(* IEC 61131-3 sources: AcpTrakStarwheel/ (part 2) *)

(* ---- StarRecovery.st ---- *)
FUNCTION_BLOCK slStarRecovery

    CASE Internal.State OF

        slREC_STATE_IDLE:
            // ----------------------------------------------------------------------- disabled

            IF Enable THEN
                Busy := 1;
                Internal.OldRemainingCount := 0;
                IF Handle = 0 THEN
                    Error := 1;
                    ErrorID := slERR_INVALID_HANDLE;
                    Internal.State := slREC_STATE_ERROR;
                ELSE
                    Internal.Handle := Handle;
                    StarInternal ACCESS Internal.Handle;
                    IF StarInternal.TypeID <> slSTAR_INTERNAL_TYPE_ID THEN
                        Error := 1;
                        ErrorID := slERR_INVALID_HANDLE;
                        Internal.State := slREC_STATE_ERROR;
                    ELSE
                        brsmemset(ADR(Internal.Data), 0, SIZEOF(Internal.Data));
                        Internal.AsmGetInfo.Assembly    := ADR(Assembly);
                        Internal.AsmGetInfo.Execute     := TRUE;
                        Internal.State := slREC_STATE_CHECK_SECTOR_SIM;
                    END_IF
                END_IF
            END_IF

        slREC_STATE_CHECK_SECTOR_SIM:

            IF Internal.AsmGetInfo.Done THEN
                Internal.SecGetShuttle.Sector := ADR(Sector);
                Internal.SecGetShuttle.Mode := mcACPTRAK_SEARCH_BACKWARD;
                Internal.SecGetShuttle.Enable := TRUE;
                Internal.State := slREC_STATE_GET_SHUTTLES;
            ELSIF Internal.AsmGetInfo.Error THEN
                Internal.AsmGetInfo.Execute := FALSE;
                Error   := TRUE;
                ErrorID := Internal.AsmGetInfo.ErrorID;
                Internal.State := slREC_STATE_ERROR;
            END_IF;

        slREC_STATE_GET_SHUTTLES:
            // ----------------------------------------------------------------------- Get shuttles in sector

            IF NOT Enable THEN
                Internal.SecGetShuttle.Next := 0;
                Internal.SecGetShuttle.Enable := 0;
                Internal.State := slREC_STATE_WAIT_NOT_BUSY;
            ELSIF Internal.SecGetShuttle.Error THEN
                Internal.SecGetShuttle.Next := 0;
                Internal.SecGetShuttle.Enable := 0;
                Error := 1;
                ErrorID := Internal.SecGetShuttle.ErrorID;
                Internal.State := slREC_STATE_ERROR;
            ELSIF Internal.SecGetShuttle.Valid AND ((Internal.SecGetShuttle.RemainingCount <> Internal.OldRemainingCount) OR (Internal.SecGetShuttle.TotalCount <= 1)) THEN
                Internal.SecGetShuttle.Next := 0;
                IF Internal.SecGetShuttle.TotalCount > 0 THEN
                    Internal.Data.Init.ShuttlePos[Internal.Data.Init.NumShuttles] := Internal.SecGetShuttle.AdditionalInfo.Position;
                    Internal.Data.Init.ShuttleAxis[Internal.Data.Init.NumShuttles] := Internal.SecGetShuttle.Axis;
                    Internal.Data.Init.NumShuttles := Internal.Data.Init.NumShuttles + 1;
                    IF Internal.AsmGetInfo.AssemblyInfo.SimulationOnPlcMode = mcACPTRAK_SIM_STATE_OFF THEN
                        Internal.State := slREC_STATE_GET_SHUTTLES_NEXT;
                    ELSIF Internal.AsmGetInfo.AssemblyInfo.SimulationOnPlcMode = mcACPTRAK_SIM_STATE_ON THEN
                        Internal.RoutedMoveAbs.Sector   := ADR(Sector);
                        Internal.RoutedMoveAbs.Axis     := ADR(Internal.SecGetShuttle.Axis);
                        Internal.RoutedMoveAbs.Position := Internal.SecGetShuttle.AdditionalInfo.Position;
                        Internal.RoutedMoveAbs.Velocity := 1.0;
                        Internal.RoutedMoveAbs.Acceleration := 20.0;
                        Internal.RoutedMoveAbs.Deceleration := 20.0;
                        Internal.RoutedMoveAbs.AdvancedParameters.StartDirection    := mcDIR_UNDEFINED;
                        Internal.RoutedMoveAbs.AdvancedParameters.EndDirection      := mcDIR_UNDEFINED;
                        Internal.RoutedMoveAbs.AdvancedParameters.ShuttleOrientation    := mcDIR_UNDEFINED;
                        Internal.RoutedMoveAbs.Execute  := TRUE;

                        Internal.State  := slREC_STATE_ATTACH_TO_SECTOR;
                    END_IF;
                ELSE //No shuttles on the sector
                    Internal.SecGetShuttle.Enable := FALSE;
                    Internal.State := slREC_STATE_DONE;
                END_IF
            END_IF

        slREC_STATE_ATTACH_TO_SECTOR:

            IF Internal.RoutedMoveAbs.Done THEN
                Internal.RoutedMoveAbs.Execute  := FALSE;
                Internal.State  := slREC_STATE_GET_SHUTTLES_NEXT;
            ELSIF Internal.RoutedMoveAbs.Error THEN
                Internal.RoutedMoveAbs.Execute  := FALSE;
                Error   := TRUE;
                ErrorID := Internal.RoutedMoveAbs.ErrorID;
                Internal.State := slREC_STATE_ERROR;
            END_IF;

        slREC_STATE_GET_SHUTTLES_NEXT:
            // -----------------------------------------------------------------------

            IF NOT Enable THEN
                Internal.SecGetShuttle.Enable := 0;
                Internal.State := slREC_STATE_WAIT_NOT_BUSY;
            ELSIF Internal.SecGetShuttle.Error THEN
                Internal.SecGetShuttle.Enable := 0;
                Error := 1;
                ErrorID := Internal.SecGetShuttle.ErrorID;
                Internal.State := slREC_STATE_ERROR;
            ELSIF Internal.SecGetShuttle.Valid THEN
                IF Internal.SecGetShuttle.RemainingCount > 0 THEN
                    Internal.OldRemainingCount := Internal.SecGetShuttle.RemainingCount;
                    Internal.SecGetShuttle.Next := TRUE;
                    Internal.State := slREC_STATE_GET_SHUTTLES;
                ELSE
                    Internal.SecGetShuttle.Enable := FALSE;
                    Internal.State := slREC_STATE_GET_USERDATA;
                END_IF
            END_IF

        slREC_STATE_RELEASE_ZONE_CHECK:
            // ----------------------------------------------------------------------- Find shuttles in the release zone

            IF Enable THEN
                IF Internal.Data.Init.ShuttlePos[Internal.Data.Init.ShuttleEvalCount] >= Parameters.MeshZoneEndPos THEN
                    Internal.State := slREC_STATE_RELEASE_ZONE_RESIZE;
                ELSE //Go to next section
                    Internal.State := slREC_STATE_MESH_ZONE_CHECK;
                END_IF;
            ELSE
                Internal.State := slREC_STATE_WAIT_NOT_BUSY;
            END_IF

        slREC_STATE_RELEASE_ZONE_RESIZE:
            // -----------------------------------------------------------------------

            IF Enable THEN
                Internal.ShResize.Axis := ADR(Internal.Data.Init.ShuttleAxis[Internal.Data.Init.ShuttleEvalCount]);
                Internal.ShResize.Command := mcACPTRAK_RESIZE_DIMENSIONS;
                Internal.ShResize.ResizeParameter := Parameters.ResizeEnd;
                Internal.ShResize.Execute := TRUE;
                Internal.State := slREC_STATE_RELEASE_ZONE_SEND;
            ELSE
                Internal.State := slREC_STATE_WAIT_NOT_BUSY;
            END_IF

        slREC_STATE_RELEASE_ZONE_SEND:
            // -----------------------------------------------------------------------

            IF NOT Enable THEN
                Internal.ShResize.Execute := 0;
                Internal.State := slREC_STATE_WAIT_NOT_BUSY;
            ELSIF Internal.ShResize.Error THEN
                Internal.ShResize.Execute := 0;
                Error := 1;
                ErrorID := Internal.ShResize.ErrorID;
                Internal.State := slREC_STATE_ERROR;
            ELSIF Internal.ShResize.Done THEN
                Internal.RoutedMoveVel.Axis := ADR(Internal.Data.Init.ShuttleAxis[Internal.Data.Init.ShuttleEvalCount]);
                Internal.RoutedMoveVel.Sector := ADR(Parameters.Release.DestinationSector);
                Internal.RoutedMoveVel.Velocity := Parameters.Release.Velocity;
                Internal.RoutedMoveVel.Acceleration := Parameters.Release.Acceleration;
                Internal.RoutedMoveVel.Deceleration := Parameters.Release.Deceleration;
                Internal.RoutedMoveVel.AdvancedParameters.StartDirection    := mcDIR_POSITIVE;
                Internal.RoutedMoveVel.AdvancedParameters.EndDirection      := mcDIR_UNDEFINED;
                Internal.RoutedMoveVel.AdvancedParameters.ShuttleOrientation    := mcDIR_UNDEFINED;

                Internal.RoutedMoveVel.Execute := TRUE;
                Internal.Data.Init.ShuttleEvalCount := Internal.Data.Init.ShuttleEvalCount + 1;
                Internal.State := slREC_STATE_RELEASE_ZONE_NEXT;
            END_IF;

        slREC_STATE_RELEASE_ZONE_NEXT:
            // ----------------------------------------------------------------------- See if there are anymore shuttles to recover

            IF NOT Enable THEN
                Internal.RoutedMoveVel.Execute := 0;
                Internal.State := slREC_STATE_WAIT_NOT_BUSY;
            ELSIF Internal.RoutedMoveVel.Error THEN
                Internal.RoutedMoveVel.Execute := 0;
                Error := 1;
                ErrorID := Internal.RoutedMoveVel.ErrorID;
                Internal.State := slREC_STATE_ERROR;
            ELSIF Internal.RoutedMoveVel.Active THEN
                Internal.RoutedMoveVel.Execute := FALSE;
                IF Internal.Data.Init.ShuttleEvalCount < Internal.Data.Init.NumShuttles THEN
                    Internal.State := slREC_STATE_RELEASE_ZONE_CHECK;
                ELSE
                    Internal.State := slREC_STATE_DONE;
                END_IF;
            END_IF

        slREC_STATE_MESH_ZONE_CHECK:
            // ----------------------------------------------------------------------- Find shuttles in the sync zone

            IF Enable THEN
                IF Internal.Data.Init.ShuttlePos[Internal.Data.Init.ShuttleEvalCount] < Parameters.MeshZoneEndPos AND
                    Internal.Data.Init.ShuttlePos[Internal.Data.Init.ShuttleEvalCount] >= (Parameters.MeshZoneStartPos) THEN
                    Internal.State := slREC_STATE_MESH_ZONE_TARGET;
                ELSE
                    //IF Parameters.SyncFurtherInEnabled THEN
                    //    Internal.Data.Sync.PocketEvalIndex    := ClosestSyncPocket(Parameters.MeshZoneStartPos, Parameters.ProcessPointStartPosition + Parameters.StartOffset, Internal.Handle);
                   // END_IF;
                    Internal.State := slREC_STATE_SYN_ZONE_CHECK;
                END_IF
            ELSE
                Internal.State := slREC_STATE_WAIT_NOT_BUSY;
            END_IF

        slREC_STATE_MESH_ZONE_TARGET:
            // ----------------------------------------------------------------------- Find the closest pocket to it and see if it is in tolerance

            //TODO: Replace with function
            //Find the closest pocket to to the shuttle
            StarInternal ACCESS Internal.Handle;
            Internal.Data.Mesh.PocketEvalIndex  := 0;
            Internal.Data.Mesh.PocketEvalIndexValid := FALSE;
            Internal.Data.Mesh.NextClosestPocketIndex   := 0;
            IF StarInternal.MaxTargetIndex > 0 THEN
                FOR Internal.i := 0 TO StarInternal.MaxTargetIndex DO
                    Internal.Data.Mesh.ShuttleErrorNew := StarInternal.PocketSync[Internal.i].TargetPosition - Internal.Data.Init.ShuttlePos[Internal.Data.Init.ShuttleEvalCount];
                    IF Internal.i = 0 THEN
                        Internal.Data.Mesh.ShuttleError := Internal.Data.Mesh.ShuttleErrorNew;
                        Internal.Data.Mesh.NextClosestPocketError := StarInternal.PocketSync[1].TargetPosition - Internal.Data.Init.ShuttlePos[Internal.Data.Init.ShuttleEvalCount];
                        Internal.Data.Mesh.NextClosestPocketIndex   := 1;
                    END_IF;
                    //Ignore any pockets that are before the sync zone
                    IF StarInternal.PocketSync[Internal.i].TargetPosition >= Parameters.ProcessPointStartPosition + Parameters.StartOffset THEN
                        Internal.Data.Mesh.PocketEvalIndexValid := TRUE;
                        IF ABS(Internal.Data.Mesh.ShuttleErrorNew) < ABS(Internal.Data.Mesh.ShuttleError) THEN
                            Internal.Data.Mesh.NextClosestPocketIndex   := Internal.Data.Mesh.PocketEvalIndex;
                            Internal.Data.Mesh.PocketEvalIndex := Internal.i;
                            Internal.Data.Mesh.NextClosestPocketError := Internal.Data.Mesh.ShuttleError;
                            Internal.Data.Mesh.ShuttleError := Internal.Data.Mesh.ShuttleErrorNew;
                        ELSIF ABS(Internal.Data.Mesh.ShuttleErrorNew) < ABS(Internal.Data.Mesh.NextClosestPocketError) AND Internal.i <> 0 THEN
                            Internal.Data.Mesh.NextClosestPocketIndex   := Internal.i;
                            Internal.Data.Mesh.NextClosestPocketError := Internal.Data.Mesh.ShuttleErrorNew;
                        END_IF
                    END_IF;
                END_FOR
            ELSE
                Error := 1;
                ErrorID := slERR_NO_TARGET;
                Internal.State := slREC_STATE_ERROR;
            END_IF

            //Check that a shuttle is not already synced with the pocket
            IF Internal.Data.Mesh.PocketEvalCount > 0 THEN
                FOR Internal.i := 0 TO Internal.Data.Mesh.PocketEvalCount - 1 DO
                    IF Internal.Data.Mesh.PocketIndices[Internal.i] = Internal.Data.Mesh.PocketEvalIndex THEN
                        Internal.Data.Mesh.ClosestPocketTaken   := TRUE;
                    ELSIF Internal.Data.Mesh.PocketIndices[Internal.i] = Internal.Data.Mesh.NextClosestPocketIndex THEN
                        Internal.Data.Mesh.NextClosestPocketTaken   := TRUE;
                    END_IF
                END_FOR
            END_IF

            //Check to see if there is another shuttle closer to this pocket, if so- try and sync to the next closest pocket
            IF NOT Internal.Data.Mesh.ClosestPocketTaken THEN
                IF Internal.Data.Mesh.ShuttleError < ABS(StarInternal.PocketSync[Internal.Data.Mesh.PocketEvalIndex].TargetPosition - Internal.Data.Init.ShuttlePos[Internal.Data.Init.ShuttleEvalCount + 1]) THEN
                    Internal.Data.Mesh.PocketIndices[Internal.Data.Mesh.PocketEvalCount] := Internal.Data.Mesh.PocketEvalIndex;
                    Internal.Data.Mesh.Axes[Internal.Data.Mesh.PocketEvalCount] := Internal.Data.Init.ShuttleAxis[Internal.Data.Init.ShuttleEvalCount];
                    Internal.State := slREC_STATE_MESH_ZONE_RESIZE;
                ELSIF NOT Internal.Data.Mesh.NextClosestPocketTaken AND (Internal.Data.Mesh.ShuttleError >= ABS(StarInternal.PocketSync[Internal.Data.Mesh.PocketEvalIndex].TargetPosition - Internal.Data.Init.ShuttlePos[Internal.Data.Init.ShuttleEvalCount + 1])) THEN
                    Internal.Data.Mesh.PocketIndices[Internal.Data.Mesh.PocketEvalCount] := Internal.Data.Mesh.NextClosestPocketIndex;
                    Internal.Data.Mesh.Axes[Internal.Data.Mesh.PocketEvalCount] := Internal.Data.Init.ShuttleAxis[Internal.Data.Init.ShuttleEvalCount];
                    Internal.State := slREC_STATE_MESH_ZONE_RESIZE;
                ELSE
                    Error := 1;
                    ErrorID := slERR_TARGET_ALREADY_SYNCED;
                    Internal.State := slREC_STATE_ERROR;
                END_IF;
            ELSIF NOT Internal.Data.Mesh.NextClosestPocketTaken THEN
                Internal.Data.Mesh.PocketIndices[Internal.Data.Mesh.PocketEvalCount] := Internal.Data.Mesh.NextClosestPocketIndex;
                Internal.Data.Mesh.Axes[Internal.Data.Mesh.PocketEvalCount] := Internal.Data.Init.ShuttleAxis[Internal.Data.Init.ShuttleEvalCount];
                Internal.State := slREC_STATE_MESH_ZONE_RESIZE;
            ELSIF Internal.Data.Mesh.NextClosestPocketTaken THEN
                Error := 1;
                ErrorID := slERR_TARGET_ALREADY_SYNCED;
                Internal.State := slREC_STATE_ERROR;
            END_IF;

        slREC_STATE_MESH_ZONE_RESIZE:
            // -----------------------------------------------------------------------

            IF Enable THEN

                Internal.ShResize.Axis := ADR(Internal.Data.Mesh.Axes[Internal.Data.Mesh.PocketEvalCount]);
                Internal.ShResize.Command := mcACPTRAK_RESIZE_DIMENSIONS;
                Internal.ShResize.ResizeParameter := Parameters.ResizeStart;
                Internal.ShResize.Execute := TRUE;

                Internal.Data.Mesh.PocketEvalCount := Internal.Data.Mesh.PocketEvalCount + 1;
                Internal.Data.Init.ShuttleEvalCount := Internal.Data.Init.ShuttleEvalCount + 1;

                Internal.State := slREC_STATE_MESH_ZONE_NEXT;
            ELSE
                Internal.State := slREC_STATE_WAIT_NOT_BUSY;
            END_IF

        slREC_STATE_MESH_ZONE_NEXT:
            // -----------------------------------------------------------------------

            IF NOT Enable THEN
                Internal.ShResize.Execute := 0;
                Internal.State := slREC_STATE_WAIT_NOT_BUSY;
            ELSIF Internal.ShResize.Error THEN
                Internal.ShResize.Execute := 0;
                Error := 1;
                ErrorID := Internal.ShResize.ErrorID;
                Internal.State := slREC_STATE_ERROR;
            ELSIF Internal.ShResize.Done THEN
                Internal.ShResize.Execute := FALSE;

                IF Internal.Data.Init.ShuttleEvalCount < Internal.Data.Init.NumShuttles THEN
                    Internal.State := slREC_STATE_MESH_ZONE_CHECK;
                ELSE
                    Internal.State := slREC_STATE_MESH_ZONE_SYNC;
                END_IF;

            END_IF;

        slREC_STATE_SYN_ZONE_CHECK:

            IF Enable THEN
                IF Internal.Data.Init.ShuttlePos[Internal.Data.Init.ShuttleEvalCount] < Parameters.MeshZoneStartPos AND
                    Internal.Data.Init.ShuttlePos[Internal.Data.Init.ShuttleEvalCount] >= (Parameters.ProcessPointStartPosition + Parameters.StartOffset) THEN
                    Internal.Data.Sync.ShuttlePos[Internal.Data.Sync.PocketEvalCount]   := Internal.Data.Init.ShuttlePos[Internal.Data.Init.ShuttleEvalCount];
                    IF NOT Internal.Data.Sync.SyncFurtherIn.ClosestPocketToMeshFound THEN
                        Internal.Data.Sync.SyncFurtherIn.ClosestPocketToMeshFound   := TRUE;
                        Internal.Data.Sync.PocketEvalIndex    := ClosestSyncPocket(Parameters.MeshZoneStartPos, Parameters.ProcessPointStartPosition + Parameters.StartOffset, Internal.Handle);
                        IF Internal.Data.Sync.PocketEvalIndex = slNO_CLOSEST_POCKET_FOUND THEN
	                        Internal.Data.Sync.SyncFurtherIn.NoClosestPocketFound   := TRUE;
                        ELSE
                            //EDGE CASE: Handles the case where a shuttle previously synced to a pocket in the mesh zone moves to the sync zone on power off. This enables the shuttle to still sync into the mesh zone
                            IF Internal.Data.Sync.PocketEvalIndex = 0 THEN
                                Internal.Data.Sync.SyncFurtherIn.FirstPocketInMeshIndex    := StarInternal.MaxTargetIndex;
                            ELSE
                                Internal.Data.Sync.SyncFurtherIn.FirstPocketInMeshIndex    := Internal.Data.Sync.PocketEvalIndex - 1;
                            END_IF;

                            IF (Internal.Data.Mesh.PocketEvalCount > 0 AND (Internal.Data.Mesh.PocketIndices[Internal.Data.Mesh.PocketEvalCount - 1] <> Internal.Data.Sync.SyncFurtherIn.FirstPocketInMeshIndex)) OR
                                Internal.Data.Mesh.PocketEvalCount = 0 THEN
                                //EDGE CASE: Still syncs a shuttle to a pocket
                                Internal.Data.Sync.SyncFurtherIn.FirstShuttleInMeshError    := ABS(StarInternal.PocketSync[Internal.Data.Sync.SyncFurtherIn.FirstPocketInMeshIndex].TargetPosition - Internal.Data.Init.ShuttlePos[Internal.Data.Init.ShuttleEvalCount]);
                                Internal.Data.Sync.SyncFurtherIn.FirstSyncPocketError       := ABS(StarInternal.PocketSync[Internal.Data.Sync.PocketEvalIndex].TargetPosition - Internal.Data.Init.ShuttlePos[Internal.Data.Init.ShuttleEvalCount]);
                                IF (Internal.Data.Sync.SyncFurtherIn.FirstShuttleInMeshError < Internal.Data.Sync.SyncFurtherIn.FirstSyncPocketError) THEN
                                    Internal.Data.Sync.PocketEvalIndex  := Internal.Data.Sync.SyncFurtherIn.FirstPocketInMeshIndex;
                                END_IF;
                            END_IF;
                        END_IF;
                    END_IF;
                    IF Internal.Data.Sync.SyncFurtherIn.NoClosestPocketFound THEN
                        Internal.State := slREC_STATE_BACKUP_ZONE_CHECK;
                    ELSE
                        Internal.State := slREC_STATE_SYN_ZONE_TARGET;
                    END_IF;
                ELSE
                    Internal.State := slREC_STATE_BACKUP_ZONE_CHECK;
                END_IF;
            ELSE
                Internal.State := slREC_STATE_WAIT_NOT_BUSY;
            END_IF;

        slREC_STATE_SYN_ZONE_TARGET:
            // ----------------------------------------------------------------------- Find the closest pocket to it and see if it is in tolerance

            IF Parameters.SyncFurtherInEnabled THEN
                IF StarInternal.PocketSync[Internal.Data.Sync.PocketEvalIndex].TargetPosition < (Parameters.ProcessPointStartPosition + Parameters.StartOffset) THEN
                    Internal.State := slREC_STATE_BACKUP_ZONE_CHECK;
                ELSE
                    Internal.Data.Sync.PocketIndices[Internal.Data.Sync.PocketEvalCount] := Internal.Data.Sync.PocketEvalIndex;
                    IF Internal.Data.Sync.PocketEvalIndex = StarInternal.MaxTargetIndex THEN
                        Internal.Data.Sync.PocketEvalIndex := 0;
                    ELSE
                        Internal.Data.Sync.PocketEvalIndex := Internal.Data.Sync.PocketEvalIndex + 1;
                    END_IF;
                    Internal.Data.Sync.Axes[Internal.Data.Sync.PocketEvalCount] := Internal.Data.Init.ShuttleAxis[Internal.Data.Init.ShuttleEvalCount];
                    Internal.State := slREC_STATE_SYN_ZONE_RESIZE;
                END_IF;
            ELSE
                //TODO: Replace with function
                //Find the closest pocket to to the shuttle
                StarInternal ACCESS Internal.Handle;
                Internal.Data.Sync.PocketEvalIndex  := 0;
                Internal.Data.Sync.PocketEvalIndexValid := FALSE;
                Internal.Data.Sync.NextClosestPocketIndex   := 0;
                IF StarInternal.MaxTargetIndex > 0 THEN
                    FOR Internal.i := 0 TO StarInternal.MaxTargetIndex DO
                        Internal.Data.Sync.ShuttleErrorNew := StarInternal.PocketSync[Internal.i].TargetPosition - Internal.Data.Init.ShuttlePos[Internal.Data.Init.ShuttleEvalCount];
                        IF Internal.i = 0 THEN
                            Internal.Data.Sync.ShuttleError := Internal.Data.Sync.ShuttleErrorNew;
                            Internal.Data.Sync.NextClosestPocketError := StarInternal.PocketSync[1].TargetPosition - Internal.Data.Init.ShuttlePos[Internal.Data.Init.ShuttleEvalCount];
                            Internal.Data.Sync.NextClosestPocketIndex   := 1;
                        END_IF;
                        //Ignore any pockets that are before the sync zone
                        IF ABS(Internal.Data.Sync.ShuttleErrorNew) < ABS(Internal.Data.Sync.ShuttleError) THEN
                            Internal.Data.Sync.NextClosestPocketIndex   := Internal.Data.Sync.PocketEvalIndex;
                            Internal.Data.Sync.PocketEvalIndex := Internal.i;
                            Internal.Data.Sync.NextClosestPocketError := Internal.Data.Sync.ShuttleError;
                            Internal.Data.Sync.ShuttleError := Internal.Data.Sync.ShuttleErrorNew;
                        ELSIF ABS(Internal.Data.Sync.ShuttleErrorNew) < ABS(Internal.Data.Sync.NextClosestPocketError) AND Internal.i <> 0 THEN
                            Internal.Data.Sync.NextClosestPocketIndex   := Internal.i;
                            Internal.Data.Sync.NextClosestPocketError := Internal.Data.Sync.ShuttleErrorNew;
                        END_IF
                    END_FOR
                ELSE
                    Error := 1;
                    ErrorID := slERR_NO_TARGET;
                    Internal.State := slREC_STATE_ERROR;
                END_IF

                //Check that a shuttle is not already synced with the pocket
                IF Internal.Data.Mesh.PocketEvalCount > 0 THEN
                    FOR Internal.i := 0 TO Internal.Data.Mesh.PocketEvalCount - 1 DO
                        IF Internal.Data.Mesh.PocketIndices[Internal.i] = Internal.Data.Sync.PocketEvalIndex THEN
                            Internal.Data.Sync.ClosestPocketTaken   := TRUE;
                        ELSIF Internal.Data.Mesh.PocketIndices[Internal.i] = Internal.Data.Sync.NextClosestPocketIndex THEN
                            Internal.Data.Sync.NextClosestPocketTaken   := TRUE;
                        END_IF
                    END_FOR
                END_IF

                //Check that a shuttle is not already synced with the pocket
                IF Internal.Data.Sync.PocketEvalCount > 0 THEN
                    FOR Internal.i := 0 TO Internal.Data.Sync.PocketEvalCount - 1 DO
                        IF Internal.Data.Sync.PocketIndices[Internal.i] = Internal.Data.Sync.PocketEvalIndex THEN
                            Internal.Data.Sync.ClosestPocketTaken   := TRUE;
                        ELSIF Internal.Data.Sync.PocketIndices[Internal.i] = Internal.Data.Sync.NextClosestPocketIndex THEN
                            Internal.Data.Sync.NextClosestPocketTaken   := TRUE;
                        END_IF
                    END_FOR
                END_IF

                //Check to see if there is another shuttle closer to this pocket, if so- try and sync to the next closest pocket
                IF NOT Internal.Data.Sync.ClosestPocketTaken THEN
                    IF StarInternal.PocketSync[Internal.Data.Sync.PocketEvalIndex].TargetPosition < Parameters.ProcessPointStartPosition + Parameters.StartOffset THEN
                        Internal.State := slREC_STATE_BACKUP_ZONE_CHECK;
                    ELSE
                        Internal.Data.Sync.PocketIndices[Internal.Data.Sync.PocketEvalCount] := Internal.Data.Sync.PocketEvalIndex;
                        Internal.Data.Sync.Axes[Internal.Data.Sync.PocketEvalCount] := Internal.Data.Init.ShuttleAxis[Internal.Data.Init.ShuttleEvalCount];
                        Internal.State := slREC_STATE_SYN_ZONE_RESIZE;
                    END_IF;
                ELSIF Internal.Data.Sync.ClosestPocketTaken AND NOT Internal.Data.Sync.NextClosestPocketTaken THEN
                    IF StarInternal.PocketSync[Internal.Data.Sync.NextClosestPocketIndex].TargetPosition < Parameters.ProcessPointStartPosition + Parameters.StartOffset THEN
                        Internal.State := slREC_STATE_BACKUP_ZONE_CHECK;
                    ELSE
                        Internal.Data.Sync.PocketIndices[Internal.Data.Sync.PocketEvalCount] := Internal.Data.Sync.NextClosestPocketIndex;
                        Internal.Data.Sync.Axes[Internal.Data.Sync.PocketEvalCount] := Internal.Data.Init.ShuttleAxis[Internal.Data.Init.ShuttleEvalCount];
                        Internal.State := slREC_STATE_SYN_ZONE_RESIZE;
                    END_IF;
                ELSIF Internal.Data.Sync.NextClosestPocketTaken THEN
                    Internal.State := slREC_STATE_BACKUP_ZONE_CHECK;
                END_IF;
            END_IF;

        slREC_STATE_SYN_ZONE_RESIZE:

            IF Enable THEN
                Internal.ShResize.Axis := ADR(Internal.Data.Sync.Axes[Internal.Data.Sync.PocketEvalCount]);
                Internal.ShResize.Command := mcACPTRAK_RESIZE_DIMENSIONS;
                Internal.ShResize.ResizeParameter := Parameters.ResizeStart;
                Internal.ShResize.Execute := TRUE;

                Internal.Data.Sync.PocketEvalCount := Internal.Data.Sync.PocketEvalCount + 1;
                Internal.Data.Init.ShuttleEvalCount := Internal.Data.Init.ShuttleEvalCount + 1;

                Internal.State := slREC_STATE_SYN_ZONE_NEXT;
            ELSE
                Internal.State := slREC_STATE_WAIT_NOT_BUSY;
            END_IF

        slREC_STATE_SYN_ZONE_NEXT:
            // -----------------------------------------------------------------------

            IF NOT Enable THEN
                Internal.ShResize.Execute := 0;
                Internal.State := slREC_STATE_WAIT_NOT_BUSY;
            ELSIF Internal.ShResize.Error THEN
                Internal.ShResize.Execute := 0;
                Error := 1;
                ErrorID := Internal.ShResize.ErrorID;
                Internal.State := slREC_STATE_ERROR;
            ELSIF Internal.ShResize.Done THEN
                Internal.ShResize.Execute := FALSE;

                IF Internal.Data.Init.ShuttleEvalCount < Internal.Data.Init.NumShuttles THEN
                    Internal.State := slREC_STATE_SYN_ZONE_CHECK;
                ELSE
                    Internal.State := slREC_STATE_MESH_ZONE_SYNC;
                END_IF;

            END_IF;

        slREC_STATE_BACKUP_ZONE_CHECK:
            // ----------------------------------------------------------------------- Look for shuttles in backup zone

            IF NOT Enable THEN
                Internal.State := slREC_STATE_WAIT_NOT_BUSY;
            ELSIF Internal.Data.Init.ShuttlePos[Internal.Data.Init.ShuttleEvalCount] >= Parameters.ProcessPointStartPosition - Parameters.ShExtentToFront THEN
                IF Internal.Data.Init.ShuttlePos[Internal.Data.Init.ShuttleEvalCount] < Parameters.ProcessPointStartPosition AND Internal.Data.Init.ShuttlePos[Internal.Data.Init.ShuttleEvalCount] >= Parameters.ProcessPointStartPosition - Parameters.ShExtentToFront THEN
                    Internal.Data.Backup.IsBeforeBarrier[Internal.Data.Backup.EvalCount]    := TRUE;
                END_IF;
                Internal.Data.Backup.Axes[Internal.Data.Backup.EvalCount] := Internal.Data.Init.ShuttleAxis[Internal.Data.Init.ShuttleEvalCount];
                Internal.Data.Backup.Positions[Internal.Data.Backup.EvalCount] := Internal.Data.Init.ShuttlePos[Internal.Data.Init.ShuttleEvalCount];
                Internal.Data.Backup.EvalCount := Internal.Data.Backup.EvalCount + 1;
                Internal.Data.Init.ShuttleEvalCount := Internal.Data.Init.ShuttleEvalCount + 1;
                IF Internal.Data.Init.ShuttleEvalCount >= Internal.Data.Init.NumShuttles THEN
                    Internal.State := slREC_STATE_MESH_ZONE_SYNC;
                END_IF;
            ELSE //Go to final recovery sequence
                Internal.State := slREC_STATE_PBACKUP_ZONE_RSIZE;
            END_IF;

        slREC_STATE_PBACKUP_ZONE_RSIZE:

            Internal.ShResize.Axis := ADR(Internal.Data.Init.ShuttleAxis[Internal.Data.Init.ShuttleEvalCount]);
            Internal.ShResize.Command := mcACPTRAK_RESIZE_DIMENSIONS;
            Internal.ShResize.ResizeParameter := Parameters.ResizeEnd;
            Internal.ShResize.Execute := TRUE;

            IF NOT Enable THEN
                Internal.ShResize.Execute := 0;
                Internal.State := slREC_STATE_WAIT_NOT_BUSY;
            ELSIF Internal.ShResize.Error THEN
                Internal.ShResize.Execute := 0;
                Error := 1;
                ErrorID := Internal.ShResize.ErrorID;
                Internal.State := slREC_STATE_ERROR;
            ELSIF Internal.ShResize.Done THEN
                Internal.ShResize.Execute := 0;
                Internal.State := slREC_STATE_PBACKUP_ZONE_SEND;
            END_IF

        slREC_STATE_PBACKUP_ZONE_SEND:
            // -----------------------------------------------------------------------

            IF Enable THEN
                Internal.ElasticMoveVel.Axis := ADR(Internal.Data.Init.ShuttleAxis[Internal.Data.Init.ShuttleEvalCount]);
                Internal.ElasticMoveVel.Velocity := Parameters.Backup.MoveToBarVelocity;
                Internal.ElasticMoveVel.Acceleration := Parameters.Backup.MoveToBarAcceleration;
                Internal.ElasticMoveVel.Deceleration := Parameters.Backup.MoveToBarDeceleration;
                Internal.ElasticMoveVel.Execute := TRUE;
                Internal.State := slREC_STATE_PBACKUP_ZONE_NEXT;
            ELSE
                Internal.State := slREC_STATE_WAIT_NOT_BUSY;
            END_IF

        slREC_STATE_PBACKUP_ZONE_NEXT:
            // -----------------------------------------------------------------------

            IF NOT Enable THEN
                Internal.ElasticMoveVel.Execute := FALSE;
                Internal.State := slREC_STATE_WAIT_NOT_BUSY;
            ELSIF Internal.ElasticMoveVel.Error THEN
                Internal.ElasticMoveVel.Execute := FALSE;
                Error := 1;
                ErrorID := Internal.ElasticMoveVel.ErrorID;
                Internal.State := slREC_STATE_ERROR;
            ELSIF Internal.ElasticMoveVel.Active THEN
                Internal.ElasticMoveVel.Execute := FALSE;
                Internal.Data.Init.ShuttleEvalCount := Internal.Data.Init.ShuttleEvalCount + 1;
                IF Internal.Data.Init.ShuttleEvalCount < Internal.Data.Init.NumShuttles THEN
                    Internal.State := slREC_STATE_PBACKUP_ZONE_RSIZE;
                ELSE
                    Internal.State := slREC_STATE_MESH_ZONE_SYNC;
                END_IF
            END_IF

        slREC_STATE_MESH_ZONE_SYNC:
            // ----------------------------------------------------------------------- Sync all of the shuttles

            StarInternal ACCESS Internal.Handle;

            IF NOT Enable THEN
                Internal.State := slREC_STATE_WAIT_NOT_BUSY;
            ELSIF Internal.Data.Mesh.RecoveredCount < Internal.Data.Mesh.PocketEvalCount THEN
                IF NOT StarInternal.PocketSync[Internal.Data.Mesh.PocketIndices[Internal.Data.Mesh.RecoveredCount]].Sync THEN
                    StarInternal.PocketSync[Internal.Data.Mesh.PocketIndices[Internal.Data.Mesh.RecoveredCount]].Axis := Internal.Data.Mesh.Axes[Internal.Data.Mesh.RecoveredCount];
                    StarInternal.PocketSync[Internal.Data.Mesh.PocketIndices[Internal.Data.Mesh.RecoveredCount]].Sync := TRUE;
                    Internal.Data.Mesh.RecoveredCount := Internal.Data.Mesh.RecoveredCount + 1;
                ELSE
                    Error := 1;
                    ErrorID := slERR_TARGET_ALREADY_SYNCED;
                    Internal.State := slREC_STATE_ERROR;
                END_IF
            ELSIF Internal.Data.Sync.PocketEvalCount <> 0 THEN
                Internal.State := slREC_STATE_SYN_ZONE_SYNC;
            ELSIF Internal.Data.Backup.EvalCount <> 0 THEN
                Internal.State := slREC_STATE_BACKUP_ZONE_TARGET;
            ELSE
                Internal.State := slREC_STATE_DONE;
            END_IF

        slREC_STATE_SYN_ZONE_SYNC:

            ReadyForStart := 1;
            IF NOT Enable THEN
                Internal.State := slREC_STATE_WAIT_NOT_BUSY;
            ELSIF Internal.Data.Sync.RecoveredCount < Internal.Data.Sync.PocketEvalCount THEN
                FOR Internal.i := 0 TO Internal.Data.Sync.PocketEvalCount - 1 DO
                    IF StarInternal.PocketSync[Internal.Data.Sync.PocketIndices[Internal.i]].TargetPosition >= Internal.Data.Sync.ShuttlePos[Internal.i] AND NOT StarInternal.PocketSync[Internal.Data.Sync.PocketIndices[Internal.i]].Sync THEN
                        StarInternal.PocketSync[Internal.Data.Sync.PocketIndices[Internal.i]].Axis := Internal.Data.Sync.Axes[Internal.i];
                        StarInternal.PocketSync[Internal.Data.Sync.PocketIndices[Internal.i]].Sync := TRUE;
                        Internal.Data.Sync.RecoveredCount   := Internal.Data.Sync.RecoveredCount + 1;
                    END_IF;
                END_FOR;
            ELSIF Internal.Data.Backup.EvalCount <> 0 THEN
                Internal.State := slREC_STATE_BACKUP_ZONE_TARGET;
            ELSE
                Internal.State := slREC_STATE_DONE;
            END_IF

        slREC_STATE_BACKUP_ZONE_TARGET:
            // ----------------------------------------------------------------------- wait for pocket to come by

            StarInternal ACCESS Internal.Handle;
            IF Internal.Data.Backup.IsBeforeBarrier[Internal.Data.Backup.RecoveredCount] THEN
                Internal.Data.Backup.PocketOvertakeIndex    := PocketOvertakeDetect(Internal.Handle, Parameters.ProcessPointStartPosition + Parameters.StartOffset);
            ELSE
                Internal.Data.Backup.PocketOvertakeIndex    := PocketOvertakeDetect(Internal.Handle, Internal.Data.Backup.Positions[Internal.Data.Backup.RecoveredCount]);
            END_IF;

            ReadyForStart := 1;

            IF NOT Enable THEN
                Internal.State := slREC_STATE_WAIT_NOT_BUSY;
            ELSIF Internal.Data.Backup.IsBeforeBarrier[Internal.Data.Backup.RecoveredCount] AND NOT Internal.Data.Backup.MovedToBarrier[Internal.Data.Backup.RecoveredCount] THEN
                Internal.BarrierCmd.Command := mcACPTRAK_BARRIER_OPEN;
                Internal.BarrierCmd.ProcessPoint    := ADR(Parameters.Backup.ProcessPointStart);
                Internal.BarrierCmd.Execute := TRUE;
                Internal.State  := slREC_STATE_BACKUP_ZONE_BAROPEN;
            ELSIF Parameters.SyncFurtherInEnabled AND NOT Internal.Data.Backup.SyncFurtherIn.SyncFurtherInFinished THEN
                Internal.Data.Backup.SyncFurtherIn.CurrentPocketIndex   := ClosestSyncPocket(Parameters.MeshZoneStartPos, Parameters.ProcessPointStartPosition + Parameters.StartOffset, Internal.Handle);
                Internal.State  := slREC_STATE_BACKUP_ZONE_SYNC_FI;
            ELSIF Internal.Data.Backup.PocketOvertakeIndex <> slNO_POCKET_DETECTED THEN
                Internal.ShResize.Axis := ADR(Internal.Data.Backup.Axes[Internal.Data.Backup.RecoveredCount]);
                Internal.ShResize.Command := mcACPTRAK_RESIZE_DIMENSIONS;
                Internal.ShResize.ResizeParameter := Parameters.ResizeStart;
                Internal.ShResize.Execute := TRUE;
                Internal.State := slREC_STATE_BACKUP_ZONE_SYNC;
            END_IF;

        slREC_STATE_BACKUP_ZONE_BAROPEN:

            IF NOT Enable THEN
                Internal.State := slREC_STATE_WAIT_NOT_BUSY;
            ELSIF Internal.BarrierCmd.Done THEN
                Internal.BarrierCmd.Execute := FALSE;
                Internal.ElasticMoveAbs.Axis    := ADR(Internal.Data.Backup.Axes[Internal.Data.Backup.RecoveredCount]);
                Internal.ElasticMoveAbs.Position    := Parameters.ProcessPointStartPosition;
                Internal.ElasticMoveAbs.Velocity    := Parameters.Backup.MoveToBarVelocity;
                Internal.ElasticMoveAbs.Acceleration    := Parameters.Backup.MoveToBarAcceleration;
                Internal.ElasticMoveAbs.Deceleration    := Parameters.Backup.MoveToBarDeceleration;
                Internal.ElasticMoveAbs.Execute := TRUE;
                Internal.State  := slREC_STATE_BACKUP_ZONE_MOVBAR;
            ELSIF Internal.BarrierCmd.Error THEN
                Internal.BarrierCmd.Execute := FALSE;
                Error := 1;
                ErrorID := Internal.BarrierCmd.ErrorID;
                Internal.State := slREC_STATE_ERROR;
            END_IF;

        slREC_STATE_BACKUP_ZONE_MOVBAR:

            IF NOT Enable THEN
                Internal.ElasticMoveAbs.Execute := FALSE;
                Internal.State := slREC_STATE_WAIT_NOT_BUSY;
            ELSIF Internal.ElasticMoveAbs.Done THEN
                Internal.ElasticMoveAbs.Execute := FALSE;
                Internal.BarrierCmd.Command := mcACPTRAK_BARRIER_CLOSE;
                Internal.BarrierCmd.ProcessPoint    := ADR(Parameters.Backup.ProcessPointStart);
                Internal.BarrierCmd.Execute := TRUE;
                Internal.State  := slREC_STATE_BACKUP_ZONE_BARCLOSE;
            ELSIF Internal.ElasticMoveAbs.CommandAborted THEN
                Internal.ElasticMoveAbs.Execute := FALSE;
                Error := 1;
                ErrorID := Internal.ElasticMoveAbs.ErrorID;
                Internal.State := slREC_STATE_ERROR;
            ELSIF Internal.ElasticMoveAbs.Error THEN
                Internal.ElasticMoveAbs.Execute := FALSE;
                Error := 1;
                ErrorID := slERR_RECOV_MOVEMNT_ABORTED;
                Internal.State := slREC_STATE_ERROR;
            END_IF;

        slREC_STATE_BACKUP_ZONE_BARCLOSE:

            IF NOT Enable THEN
                Internal.BarrierCmd.Execute := FALSE;
                Internal.State := slREC_STATE_WAIT_NOT_BUSY;
            ELSIF Internal.BarrierCmd.Done THEN
                Internal.BarrierCmd.Execute := FALSE;
                Internal.Data.Backup.MovedToBarrier[Internal.Data.Backup.RecoveredCount]    := TRUE;
                Internal.State  := slREC_STATE_BACKUP_ZONE_TARGET;
            ELSIF Internal.BarrierCmd.Error THEN
                Internal.BarrierCmd.Execute := FALSE;
                Error := 1;
                ErrorID := Internal.BarrierCmd.ErrorID;
                Internal.State := slREC_STATE_ERROR;
            END_IF;

        slREC_STATE_BACKUP_ZONE_SYNC:
            // -----------------------------------------------------------------------

            StarInternal ACCESS Internal.Handle;

            IF NOT Enable THEN
                Internal.ShResize.Execute := FALSE;
                Internal.State := slREC_STATE_WAIT_NOT_BUSY;
            ELSIF Internal.ShResize.Error THEN
                Internal.ShResize.Execute := 0;
                Error := 1;
                ErrorID := Internal.ShResize.ErrorID;
                Internal.State := slREC_STATE_ERROR;
            ELSIF Internal.ShResize.Done THEN
                Internal.ShResize.Execute := 0;
                IF StarInternal.PocketSync[Internal.Data.Backup.PocketOvertakeIndex].Sync THEN
                    Error := 1;
                    ErrorID := slERR_TARGET_ALREADY_SYNCED;
                    Internal.State := slREC_STATE_ERROR;
                ELSE
                    StarInternal.PocketSync[Internal.Data.Backup.PocketOvertakeIndex].Axis := Internal.Data.Backup.Axes[Internal.Data.Backup.RecoveredCount];
                    StarInternal.PocketSync[Internal.Data.Backup.PocketOvertakeIndex].Sync := 1;
                    Internal.Data.Backup.RecoveredCount := Internal.Data.Backup.RecoveredCount + 1;
                    IF Internal.Data.Backup.RecoveredCount < Internal.Data.Backup.EvalCount THEN
                        Internal.State := slREC_STATE_BACKUP_ZONE_TARGET;
                    ELSE
                        Internal.State := slREC_STATE_DONE;
                    END_IF
                END_IF
            END_IF

        slREC_STATE_BACKUP_ZONE_SYNC_FI:

            StarInternal ACCESS Internal.Handle;

            IF (Internal.Data.Backup.SyncFurtherIn.CurrentPocketIndex <> slNO_CLOSEST_POCKET_FOUND) AND (Internal.Data.Backup.RecoveredCount <> Internal.Data.Backup.EvalCount) THEN
                StarInternal.PocketSync[Internal.Data.Backup.SyncFurtherIn.CurrentPocketIndex].Axis := Internal.Data.Backup.Axes[Internal.Data.Backup.RecoveredCount];
                StarInternal.PocketSync[Internal.Data.Backup.SyncFurtherIn.CurrentPocketIndex].Sync := TRUE;
                Internal.Data.Backup.RecoveredCount := Internal.Data.Backup.RecoveredCount + 1;
                Internal.State  := slREC_STATE_BACKUP_ZONE_TARGET;
            ELSE
                Internal.Data.Backup.SyncFurtherIn.SyncFurtherInFinished    := TRUE;
                IF Internal.Data.Backup.RecoveredCount < Internal.Data.Backup.EvalCount THEN
                    Internal.State := slREC_STATE_BACKUP_ZONE_TARGET;
                ELSE
                    Internal.State := slREC_STATE_DONE;
                END_IF
            END_IF;

        slREC_STATE_GET_USERDATA:

            // populates buffer so USERDATA_SET doesn't overwrite other parameters
            Internal.ShCopyUserData.Axis := ADR(Internal.Data.Init.ShuttleAxis[Internal.Data.UserData.UserDataWriteCount]);
            Internal.ShCopyUserData.DataAddress := Parameters.UserData.UserDataAddress;
            Internal.ShCopyUserData.DataSize := Parameters.UserData.UserDataSize;
            Internal.ShCopyUserData.Mode := mcACPTRAK_USERDATA_GET;
            Internal.ShCopyUserData.Execute := TRUE;

            IF Internal.ShCopyUserData.Error THEN
                Internal.ShCopyUserData.Execute := FALSE;
                Error := 1;
                ErrorID := Internal.ShCopyUserData.ErrorID;
                Internal.State := slREC_STATE_ERROR;
            ELSIF Internal.ShCopyUserData.Done THEN
                Internal.ShCopyUserData.Execute	:= FALSE;

                IF Parameters.UserData.UserDataAddress = 0 OR
                    Parameters.UserData.UserDataSize = 0 OR
                    Parameters.UserData.SrcUserDataWriteAddress = 0 OR
                    Parameters.UserData.DstUserDataWriteAddress = 0 OR
                    Parameters.UserData.UserDataWriteSize = 0 THEN

                    Error := 1;
                    ErrorID := slERR_INVALID_USER_DATA;
                    Internal.State := slREC_STATE_ERROR;

                ELSE

                    brsmemcpy(Parameters.UserData.DstUserDataWriteAddress, Parameters.UserData.SrcUserDataWriteAddress, Parameters.UserData.UserDataWriteSize);
                    Internal.State := slREC_STATE_SET_USERDATA;

                END_IF

            END_IF

        slREC_STATE_SET_USERDATA:

            StarInternal ACCESS Internal.Handle;

            Internal.ShCopyUserData.Axis := ADR(Internal.Data.Init.ShuttleAxis[Internal.Data.UserData.UserDataWriteCount]);
            Internal.ShCopyUserData.DataAddress := Parameters.UserData.UserDataAddress;
            Internal.ShCopyUserData.DataSize := Parameters.UserData.UserDataSize;
            Internal.ShCopyUserData.Mode := mcACPTRAK_USERDATA_SET;
            Internal.ShCopyUserData.Execute := TRUE;

            IF Internal.ShCopyUserData.Error THEN
                Internal.ShCopyUserData.Execute := FALSE;
                Error := 1;
                ErrorID := Internal.ShCopyUserData.ErrorID;
                Internal.State := slREC_STATE_ERROR;
            ELSIF Internal.ShCopyUserData.Done THEN
                Internal.ShCopyUserData.Execute	:= FALSE;
                Internal.Data.UserData.UserDataWriteCount := Internal.Data.UserData.UserDataWriteCount + 1;
                IF Internal.Data.UserData.UserDataWriteCount < Internal.Data.Init.NumShuttles THEN
                    Internal.State := slREC_STATE_GET_USERDATA;
                ELSE
                    Internal.State := slREC_STATE_RELEASE_ZONE_CHECK;
                END_IF

            END_IF

        slREC_STATE_DONE:

            Done := 1;
            ReadyForStart := 1;

            IF NOT Enable THEN
                ReadyForStart := 0;
                Done:= 0;
                Internal.State := slREC_STATE_WAIT_NOT_BUSY;
            END_IF

        slREC_STATE_WAIT_NOT_BUSY:

            IF NOT Internal.SecGetShuttle.Busy OR Internal.ShResize.Busy OR Internal.RoutedMoveVel.Busy OR Internal.ElasticMoveVel.Busy OR Internal.ShCopyUserData.Busy THEN
                Busy := 0;
                Internal.State := slREC_STATE_IDLE;
            END_IF

        slREC_STATE_ERROR:

            ReadyForStart := 0;

            IF NOT Enable THEN
                Error := 0;
                ErrorID := ERR_OK;
                Internal.State := slREC_STATE_WAIT_NOT_BUSY;
            END_IF

    END_CASE

    Internal.SecGetShuttle();
    Internal.ShResize();
    Internal.RoutedMoveVel();
    Internal.ElasticMoveVel();
    Internal.ElasticMoveAbs();
    Internal.ShCopyUserData();
    Internal.BarrierCmd();
    Internal.AsmGetInfo();
    Internal.RoutedMoveAbs();

END_FUNCTION_BLOCK

(* ---- StarSync.st ---- *)
FUNCTION_BLOCK slStarSync

    //Check for an error on a pocket
    Internal.PocketSyncError := 0;
    Internal.PocketSyncErrorID := ERR_OK;
    FOR Internal.i := 0 TO slMAX_TARGET_IDX DO
        IF Internal.PocketSync[Internal.i].Error THEN
            Internal.PocketSyncError := 1;
            Internal.PocketSyncErrorID := Internal.PocketSync[Internal.i].ErrorID;
            EXIT;
        END_IF
    END_FOR

    IF Enable AND Busy THEN
        // Continuously watch for calculated Track Sync Positions to overtake the Sync Threshold, and update the NextSyncTarget selector
        // Also monitor for completion
        FOR Internal.i := 0 TO Internal.MaxTargetIndex DO
            IF Internal.PocketSync[Internal.i].TargetPosition >= Parameters.Buffer.StagingPosition + Parameters.StartOffset AND
                Internal.LastTargetPosition[Internal.i] < Parameters.Buffer.StagingPosition + Parameters.StartOffset AND
                Internal.PocketSync[Internal.i].TargetPosition < Parameters.SyncPar.StarCalcTarget.SectorTangentPos AND
                Internal.PocketSync[Internal.i].Active AND
                NOT Internal.PocketSync[Internal.i].Sync
                AND Internal.RecoveryDone THEN

                Internal.PocketDisabled := 0;
                IF DisablePockets AND (Parameters.Skip.NumDisabled > 0) THEN
					FOR Internal.n := 0 TO MIN(Parameters.Skip.NumDisabled - 1, slMAX_DISABLE_POCKET_IDX) DO
                        IF Parameters.Skip.DisabledIdx[Internal.n] = (Internal.i MOD (Parameters.SyncPar.StarCalcTarget.StarwheelPocketCount)) THEN
                            Internal.PocketDisabled := 1;
                            EXIT;
                        END_IF
                    END_FOR
				END_IF

				IF Internal.PocketDisabled THEN
					Internal.NewDisabledOvertake	:= TRUE;
				ELSE
					Internal.NextSyncTarget			:= Internal.i;
					Internal.NewOvertakeDetected	:= TRUE;
				END_IF;

            END_IF
            IF Internal.PocketSync[Internal.i].Done THEN
                Internal.PocketSync[Internal.i].Sync := 0;
            END_IF
        END_FOR
    ELSE
        Internal.NextSyncTarget := 0;
        Internal.NewOvertakeDetected := FALSE;
    END_IF

    CASE Internal.State OF

        slSTAR_STATE_INIT:

            Handle := ADR(Internal);
            Internal.TypeID := slSTAR_INTERNAL_TYPE_ID;
            Internal.State := slSTAR_STATE_IDLE;

        slSTAR_STATE_IDLE:

            IF Enable THEN

                Busy := 1;

                // Calculate how many periods of starwheel rotation we should calculate track positions for,
                // in order to cover the area from SyncPP TO ReleasePP
                Internal.PeriodCount := 0;
                FOR Internal.i := 0 TO slMAX_PERIOD_IDX DO
                    IF Internal.i * brmTWOPI * Parameters.SyncPar.StarCalcTarget.StarwheelRadius > (Parameters.SyncPar.StarCalcTarget.SectorTangentPos - Parameters.StartOffset) THEN
                        Internal.PeriodCount := UINT_TO_USINT(Internal.i + 1);
                        EXIT;
                    END_IF
                END_FOR

                Internal.MaxTargetIndex := Parameters.SyncPar.StarCalcTarget.StarwheelPocketCount * Internal.PeriodCount - 1;

                IF Internal.MaxTargetIndex > slMAX_TARGET_IDX THEN

                    Error := 1;
                    ErrorID := slERR_MAX_TARGET_IDX;
                    Internal.State := slSTAR_STATE_RESET_FB;

                ELSE

                    Internal.PocketWidth        := brmTWOPI * Parameters.SyncPar.StarCalcTarget.StarwheelRadius / USINT_TO_REAL(Parameters.SyncPar.StarCalcTarget.StarwheelPocketCount);
                    Internal.MeshZoneStartPos   := Parameters.SyncPar.StarCalcTarget.SectorTangentPos - Internal.PocketWidth*0.75;
                    Internal.MeshZoneEndPos     := Parameters.SyncPar.StarCalcTarget.SectorTangentPos + Internal.PocketWidth;

                    brsmemset(ADR(Internal.Buffer), 0, SIZEOF(Internal.Buffer));
                    Internal.StarBuffer.Buffer := ADR(Internal.Buffer);
                    Internal.StarBuffer.ProcessPoint := ADR(ProcessPointStart);
                    Internal.StarBuffer.Parameters := ADR(Parameters.Buffer);

                    FOR Internal.i := 0 TO slMAX_TARGET_IDX  DO
                        Internal.PocketSync[Internal.i].TargetIndex := UINT_TO_USINT(Internal.i);
                        Internal.PocketSync[Internal.i].PeriodCount := Internal.PeriodCount;
                        Internal.PocketSync[Internal.i].Parameters := ADR(Parameters.SyncPar);
                        Internal.PocketSync[Internal.i].CalcData := ADR(Internal.StarCalcData);
                        Internal.PocketSync[Internal.i].Enable := (Internal.i <= Internal.MaxTargetIndex);
                    END_FOR

                    Internal.State := slSTAR_STATE_RECOVER;

                END_IF

            END_IF

        slSTAR_STATE_RECOVER:

            Internal.RecoveryPar.MeshZoneStartPos   := Internal.MeshZoneStartPos;
            Internal.RecoveryPar.SyncFurtherInEnabled   := Parameters.Recovery.SyncFurtherInEnabled;
            Internal.RecoveryPar.MeshZoneEndPos     := Internal.MeshZoneEndPos;
            Internal.RecoveryPar.SectorTangentPos   := Parameters.SyncPar.StarCalcTarget.SectorTangentPos;
            Internal.RecoveryPar.ShExtentToFront        := Parameters.ShExtentToFront;
            Internal.RecoveryPar.ProcessPointStartPosition := Parameters.Buffer.StagingPosition;
            Internal.RecoveryPar.StartOffset := Parameters.StartOffset;
            Internal.RecoveryPar.ResizeStart := Parameters.SyncPar.ResizeStart;
            Internal.RecoveryPar.ResizeEnd := Parameters.SyncPar.ResizeEnd;
            Internal.RecoveryPar.Release.Position := Parameters.SyncPar.Release.Position;
            Internal.RecoveryPar.Release.DestinationSector := Parameters.Recovery.Release.DestinationSector;
            Internal.RecoveryPar.Release.Velocity := Parameters.Recovery.Release.Velocity;
            Internal.RecoveryPar.Release.Acceleration := Parameters.Recovery.Release.Acceleration;
            Internal.RecoveryPar.Release.Deceleration := Parameters.Recovery.Release.Deceleration;
            Internal.RecoveryPar.UserData := Parameters.Recovery.UserData;
            Internal.RecoveryPar.PocketErrorTolerance := Parameters.Recovery.PocketErrorTolerance;
            Internal.RecoveryPar.Backup.ProcessPointStart := ProcessPointStart;
            Internal.RecoveryPar.Backup.BackupTolerance := Parameters.Recovery.BackupTolerance;
            Internal.RecoveryPar.Backup.MoveToBarVelocity   := Parameters.Recovery.MoveToBarVelocity;
            Internal.RecoveryPar.Backup.MoveToBarAcceleration   := Parameters.Recovery.MoveToBarAcceleration;
            Internal.RecoveryPar.Backup.MoveToBarDeceleration   := Parameters.Recovery.MoveToBarDeceleration;

            Internal.Recovery.Parameters := ADR(Internal.RecoveryPar);
            Internal.Recovery.Sector := ADR(Sector);
            Internal.Recovery.Handle := Handle;
            Internal.Recovery.Assembly  := ADR(Assembly);
            Internal.Recovery.Enable := 1;

            IF Internal.Recovery.ReadyForStart THEN
                ReadyForStart := 1;
            END_IF;

            IF NOT Enable THEN
                Internal.State := slSTAR_STATE_RESET_FB;
            ELSIF Internal.Recovery.Error THEN
                Error := 1;
                ErrorID := Internal.Recovery.ErrorID;
                Internal.State := slSTAR_STATE_RESET_FB;
            ELSIF Internal.Recovery.Done THEN
                ReadyForStart := 1;
                Internal.RecoveryDone   := TRUE;
                Internal.Recovery.Enable := 0;
                Internal.StarBuffer.Enable := 1;
                Active := 1;
                Internal.NextSyncFITarget   := ClosestSyncPocket(Internal.MeshZoneStartPos, Parameters.Buffer.StagingPosition + Parameters.StartOffset, Handle);
                Internal.State := slSTAR_STATE_WAIT_TARGET;
            END_IF

        slSTAR_STATE_WAIT_TARGET:

            IF NOT Enable THEN
                Internal.State := slSTAR_STATE_RESET_FB;
            ELSIF Internal.StarBuffer.Error THEN
                Error := 1;
                ErrorID := Internal.StarBuffer.ErrorID;
                Internal.State := slSTAR_STATE_RESET_FB;
            ELSIF Internal.PocketSyncError THEN
                Error := 1;
                ErrorID := Internal.PocketSyncErrorID;
                Internal.State := slSTAR_STATE_RESET_FB;
                //Check for new pocket
            ELSIF Internal.NewOvertakeDetected THEN
                IF SkipPockets THEN
                    IF Internal.SkipCount < Parameters.Skip.NumSkips THEN
                        Internal.NewOvertakeDetected := 0;
                        Internal.SkipCount := Internal.SkipCount + 1;
                    ELSE
                        Internal.State := slSTAR_STATE_WAIT_SHUTTLE;
                        Internal.SkipCount := 0;
                    END_IF
                ELSE
                    Internal.State := slSTAR_STATE_WAIT_SHUTTLE;
				END_IF
            END_IF

        slSTAR_STATE_WAIT_SHUTTLE:

            IF NOT Enable THEN
                Internal.State := slSTAR_STATE_RESET_FB;
            ELSIF Internal.StarBuffer.Error THEN
                Error := 1;
                ErrorID := Internal.StarBuffer.ErrorID;
                Internal.State := slSTAR_STATE_RESET_FB;
            ELSIF Internal.Buffer.ReadIdx <> Internal.Buffer.WriteIdx THEN
                Internal.State := slSTAR_STATE_SYNC;
            END_IF

        slSTAR_STATE_SYNC:

            IF Parameters.Recovery.SyncFurtherInEnabled AND NOT Internal.SyncFurtherInDone THEN
                Internal.PocketSync[Internal.NextSyncFITarget].Axis := Internal.Buffer.Shuttles[Internal.Buffer.ReadIdx];
                Internal.PocketSync[Internal.NextSyncFITarget].Sync := 1;
                Internal.NextSyncFITarget   := ClosestSyncPocket(Internal.MeshZoneStartPos, Parameters.Buffer.StagingPosition + Parameters.StartOffset, Handle);
                IF Internal.NextSyncFITarget = slNO_CLOSEST_POCKET_FOUND THEN
                    Internal.SyncFurtherInDone  := TRUE;
                    Internal.NewOvertakeDetected := 0;
                END_IF
            ELSE
                Internal.PocketSync[Internal.NextSyncTarget].Axis := Internal.Buffer.Shuttles[Internal.Buffer.ReadIdx];
                Internal.PocketSync[Internal.NextSyncTarget].Sync := 1;
                Internal.NewOvertakeDetected := 0;
                Internal.State := slSTAR_STATE_WAIT_TARGET;
            END_IF
            Internal.Buffer.ReadIdx := (Internal.Buffer.ReadIdx + 1) MOD (slMAX_SH_IDX_IN_SEC + 1);
            Internal.State := slSTAR_STATE_WAIT_TARGET;

        slSTAR_STATE_RESET_FB:

            Active := 0;
            ReadyForStart := 0;
            Internal.NextSyncTarget := 0;
            Internal.NewOvertakeDetected := 0;
            Internal.StarBuffer.Enable := 0;
            Internal.Recovery.Enable := 0;
            Internal.SyncFurtherInDone  := FALSE;
            Internal.RecoveryDone   := FALSE;
            Internal.ErrorID := ErrorID;
            FOR Internal.i := 0 TO slMAX_TARGET_IDX DO
                Internal.PocketSync[Internal.i].Sync := 0;
                Internal.PocketSync[Internal.i].Enable := 0;
            END_FOR
            IF Error THEN
                Internal.State := slSTAR_STATE_ERROR;
            ELSE
                //We only get here if the enable has been dropped
                Internal.State := slSTAR_STATE_WAIT_NOT_BUSY;
            END_IF

        slSTAR_STATE_WAIT_NOT_BUSY:

            Internal.PocketSyncBusy := 0;
            FOR Internal.i := 0 TO slMAX_TARGET_IDX DO
                IF Internal.PocketSync[Internal.i].Busy THEN
                    Internal.PocketSyncBusy := 1;
                END_IF
            END_FOR

            IF NOT (Internal.PocketSyncBusy OR Internal.StarBuffer.Busy OR Internal.Recovery.Busy) THEN
                Error := 0;
                ErrorID := ERR_OK;
                Busy := 0;
                Internal.State := slSTAR_STATE_IDLE;
            END_IF

        slSTAR_STATE_ERROR:

            IF NOT Enable THEN
                Error := 0;
                ErrorID := ERR_OK;
                Internal.State := slSTAR_STATE_WAIT_NOT_BUSY;
            END_IF

	END_CASE

	IF Enable THEN
		IF Parameters.SyncPar.StarCalcTarget.StarwheelPeriod <> 0 THEN
			//Calculate latency compensation
			Internal.StarCalcData.StarPosPredict := StarwheelPosition + StarwheelVelocity * TIME_TO_REAL(Parameters.SyncPar.StarCalcTarget.DeltaT) / 1000.0;
			Internal.StarCalcData.StarPosPredict := EuclideanModuloFLT(Internal.StarCalcData.StarPosPredict, Parameters.SyncPar.StarCalcTarget.StarwheelPeriod);
		END_IF

		//Detect starwheel position rollover
		IF (Internal.StarCalcData.StarPosPredict - Internal.OldStarPosPredict) > (Parameters.SyncPar.StarCalcTarget.StarwheelPeriod / 4.0) THEN //Rollover backwards
			Internal.StarCalcData.CurrentStarwheelPeriod := Internal.StarCalcData.CurrentStarwheelPeriod - 1;
		ELSIF (Internal.OldStarPosPredict - Internal.StarCalcData.StarPosPredict) > (Parameters.SyncPar.StarCalcTarget.StarwheelPeriod / 4.0) THEN //Rollover forwards
			Internal.StarCalcData.CurrentStarwheelPeriod := Internal.StarCalcData.CurrentStarwheelPeriod + 1;
		END_IF

		// Constrain CurrentStarwheelPeriod to {0..Sector.Par.PeriodCount-1}, EuclideanModulo deals with negatives correctly versus standard truncated form
		Internal.StarCalcData.CurrentStarwheelPeriod := EuclideanModuloINT(Internal.StarCalcData.CurrentStarwheelPeriod, Internal.PeriodCount);
		Internal.StarCalcData.MultiturnPosition := Internal.StarCalcData.StarPosPredict + (INT_TO_REAL(Internal.StarCalcData.CurrentStarwheelPeriod) * Parameters.SyncPar.StarCalcTarget.StarwheelPeriod);
	END_IF

	//Capture old starwheel predict position
	Internal.OldStarPosPredict := Internal.StarCalcData.StarPosPredict;

    Internal.StarBuffer();
    Internal.Recovery();
    FOR Internal.i := 0 TO slMAX_TARGET_IDX DO
        Internal.LastTargetPosition[Internal.i] := Internal.PocketSync[Internal.i].TargetPosition;
        Internal.PocketSync[Internal.i]();
        //Initialize the last target position so that the system
        //does not think that targets have just passed the sync point
        IF Internal.PocketSync[Internal.i].Active AND NOT Internal.LastPocketActiveState[Internal.i] THEN
            Internal.LastTargetPosition[Internal.i] := Internal.PocketSync[Internal.i].TargetPosition;
        END_IF
        Internal.LastPocketActiveState[Internal.i] := Internal.PocketSync[Internal.i].Active;
    END_FOR

END_FUNCTION_BLOCK

(* ---- Constants.var ---- *)
(*Errors*)
VAR CONSTANT
	slERR_ZERO_PERIOD : DINT := -5000; (*The period is zero and thus invalid*)
	slERR_ZERO_POCKETS : DINT := -5001; (*The number of pockets are zero and thus invalid*)
	slERR_POCKET_GT_COUNT : DINT := -5002; (*The target pocket is greater than the pocket count*)
	slERR_ZERO_RADIUS : DINT := -5003; (*The starwheel radius cannot be zero*)
	slERR_INVALID_HANDLE : DINT := -5004; (*The handle provided is invalid*)
	slERR_MAX_TARGET_IDX : DINT := -5005; (*The maximum target index is too large*)
	slERR_NO_TARGET : DINT := -5006; (*No targets available*)
	slERR_TARGET_ALREADY_SYNCED : DINT := -5007; (*Attempted to sync to a target that is already synced*)
	slERR_TARGET_OUT_OF_TOL : DINT := -5008; (*Sync target is out of tolerance from shuttle position*)
	slERR_INVALID_USER_DATA : DINT := -5009; (*Invalid user data parameters*)
	slERR_SYNC_ABORTED : DINT := -5010; (*The synchronization was aborted while a shuttle was in sync*)
	slERR_RECOV_MOVEMNT_ABORTED : DINT := -5011;
	slERR_MAX_STAR_SH_IDX : DINT := -5111; (*Index of shuttle on star sector exceeds limit*)
END_VAR
(*Values*)
VAR CONSTANT
	slNO_POCKET_DETECTED : UINT := 65535;
	slNO_CLOSEST_POCKET_FOUND : UINT := 65535; (*No closest pocket was found (sync further in functionality)*)
	slMAX_TARGET_IDX : UINT := 64; (*Maximum target index*)
	slMAX_SH_IDX_IN_SEC : UINT := 64; (*Maximum shuttle index in sector*)
	slMAX_PERIOD_IDX : USINT := 32; (*Maximum period index to track targets through*)
	slMAX_DISABLE_POCKET_IDX : USINT := 24; (*Maximum index of pocket to disable*)
	slMAX_STATE_TRACE_IDX : USINT := 100; (*Maximum index of the state trace*)
	slSTAR_INTERNAL_TYPE_ID : UDINT := 648661409; (*ID to indicate that structure is StarSync Internal Data*)
END_VAR
